FUNCTION "Strip Sign" : String
{ S7_Optimized_Access := 'TRUE' }
VERSION : 0.1
   VAR_INPUT
      "string" : String;
   END_VAR

   VAR_TEMP
      Length : Int;
      "String Box" : String;
      "Test Character" : String;
   END_VAR

   VAR CONSTANT
      "+" : Char := '+';
      "-" : Char := '-';
   END_VAR


BEGIN
	#"String Box" := #string;
	#"Test Character" := LEFT_STRING(IN := #"String Box",
	                                  L := 1);
	IF #"Test Character" = #"+" OR #"Test Character" = #"-" THEN
	    #Length := LEN(#"String Box");
	    #"String Box" := RIGHT_STRING(IN := #"String Box", L := #Length - 1);

	END_IF;
	#"Strip Sign" := #"String Box";
END_FUNCTION

